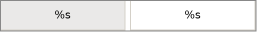
VISUALIZATION VISU_ConfigStringEntry  // 257x32
VAR_IN_OUT
    active : STRING;
    editable : STRING;
END_VAR
    Textfield (0,0 125x30), "%s", text variable: active, input disabled if: TRUE
    Textfield (130,0 125x30), "%s", text variable: editable, colour toggle: editable <> active
        OnMouseClick: write the text variable via Default
END_VISUALIZATION

(* stored: Version 1.1.0.1, ProductVersion 3.1.0.36
   Visu VISU_ConfigStringEntry: Id {e02bd99e-2e2b-4af3-b422-212854be0bf2} *)
